(* IEC 61131-3 sources: SRCI/RobotLibrary/Library/POUs/_internal/BaseFBs, 4 files *)

(* ---- RobotLibraryBaseEnableFB.st ---- *)
FUNCTION_BLOCK RobotLibraryBaseEnableFB EXTENDS RobotLibraryBaseFB
// -------------------------------------------------------------------------
//  SRCI Robot Library
// -------------------------------------------------------------------------
//
//  Object:      RobotLibraryBaseFB
//  Author:      Thorsten Brach
//  Date:        2024-08-11
//
//  Description:
//
//
//  Copyright:
//    (C) 2024 Thorsten Brach. All rights reserved
//             Licensed under the LGPL-3.0 license.
//
//  Disclaimer:
//    This project is provided without any guarantee and can be used for
//    private and commercial purposes. Any use is at the user’s
//    own risk and responsibility.
//
// -------------------------------------------------------------------------
VAR_INPUT
  /// Set TRUE to activate / Set False to deactivate
  Enable            : BOOL;
END_VAR

VAR_OUTPUT
  /// FB is being processed
  Busy              : BOOL;
  /// TRUE while function is active
  Enabled           : BOOL;
END_VAR

VAR
  /// Rising edge for enable
  {attribute 'hide'}
 _enable_R          : R_TRIG;
  /// Falling edge for enable
  {attribute 'hide'}
 _enable_F          : F_TRIG;
END_VAR

  SUPER^(AxesGroup := AxesGroup);

END_FUNCTION_BLOCK

METHOD PROTECTED OnCall
VAR_IN_OUT
  /// Robot assignment of function
  AxesGroup : AxesGroup;
END_VAR

VAR
  /// internal return value
 _retVal : DINT;
END_VAR

  SUPER^.OnCall(AxesGroup := AxesGroup);

  // building rising and falling edges
  _enable_R( CLK := Enable);
  _enable_F( CLK := Enable);

  // Check command execution is allowed ?
  IF ((     Enable                                 ) AND
      ( NOT AxesGroup.State.Initialized            ) AND
      ( NOT AxesGroup.State.Synchronized           ) AND
      (     MyType <> 'MC_ExchangeConfigurationFB' ) AND // is part of init sequence
      (     MyType <> 'MC_ReadMessagesFB'          ) AND // is part of init sequence
      (     MyType <> 'MC_ReadRobotDataFB'         ))    // is part of init sequence
  THEN
    ErrorID := RobotLibraryErrorIdEnum.ERR_COMMANDS_NOT_ENABLED;
    Error   := TRUE;
    Busy    := FALSE;
  END_IF

  // On execution started
  IF ( _enable_R.Q )
  THEN
    OnExecStart(AxesGroup := AxesGroup);
  END_IF

  // On execution cancel
  IF ( Busy ) AND ( _enable_F.Q )
  THEN
    // set cancel flag
   _cancel := TRUE;
  END_IF

  IF ( _cancel )
  THEN
    // call Cancel
   _retVal := OnExecCancel(AxesGroup := AxesGroup);

    // done or error ?
    IF ( _retVal <> RobotLibraryConstants.RUNNING )
    THEN
      // reset cancel flag
     _cancel := FALSE;
  	END_IF
  END_IF

  // On execution error clear
  IF ( Error ) AND ( _enable_F.Q )
  THEN
    // set ClearError flag
   _clearError := TRUE;
  END_IF

  IF ( _clearError )
  THEN
   _retVal := OnExecErrorClear(AxesGroup := AxesGroup);

    // done or error ?
    IF ( _retVal <> RobotLibraryConstants.RUNNING )
    THEN
      // reset ClearError flag
     _clearError := FALSE;
  	END_IF
  END_IF

END_METHOD

METHOD Protected OnExecCancel : DINT
VAR_IN_OUT
  /// Robot assignment of function
  AxesGroup : AxesGroup;
END_VAR
VAR
  /// internal return value
 _retVal    : DINT;
END_VAR

  OnExecCancel := Reset();

  // Create log entry
  CreateLogMessagePara1 ( Timestamp   := AxesGroup.State.SystemTime,
                          MessageType := MessageType.CMD,
                          Severity    := Severity.DEBUG,
                          MessageCode := 0,
                          MessageText := 'Execution of {1} cancled ',
                          Para1       := MyType);

  // try to remove cmd
  _retVal := AxesGroup.Acyclic.ActiveCommandRegister.RemoveCmd(_uniqueID);

  IF (_retVal = RobotLibraryConstants.OK)
  THEN
    // Create log entry
    CreateLogMessagePara1 ( Timestamp   := AxesGroup.State.SystemTime,
                            MessageType := MessageType.CMD,
                            Severity    := Severity.DEBUG,
                            MessageCode := 0,
                            MessageText := '{1} successfully removed from ACR',
                            Para1       := MyType);
  ELSE
    // Create log entry
    CreateLogMessagePara1 ( Timestamp   := AxesGroup.State.SystemTime,
                            MessageType := MessageType.CMD,
                            Severity    := Severity.DEBUG,
                            MessageCode := 0,
                            MessageText := '{1} was not removed from ACR because execution was already in progress',
                            Para1       := MyType);
  END_IF

END_METHOD

METHOD PROTECTED OnExecErrorClear : DINT
VAR_IN_OUT
  /// Robot assignment of function
  AxesGroup : AxesGroup;
END_VAR

  OnExecErrorClear := RobotLibraryConstants.RUNNING;

  CASE _stepClearError OF

    0:  // Reset
        Reset();
        // trigger parameter update to disable FB
       _parameterUpdateInternal := TRUE;
        // call Check Parameter changed method to trigger the parameter update to deactivate jogging mode
        CheckParameterChanged(AxesGroup := AxesGroup);
        // set timeout
        SetTimeout(PT := _timeoutClearError, rTimer := _timerClearError);
        // inc step counter
       _stepClearError := _stepClearError + 1;

    1: IF ( _responseReceived )
       THEN
         // reset response received flag
        _responseReceived := FALSE;
         // reset step counter
        _stepClearError := 0;
         // finished
         OnExecErrorClear := RobotLibraryConstants.OK;
       ELSE
         // timeout exceeded ?
         IF (CheckTimeout(_timerClearError) = RobotLibraryConstants.OK)
         THEN
           OnExecErrorClear := RobotLibraryConstants.HAS_ERROR;
         END_IF
  	   END_IF
  ELSE
    // invalid step
    ErrorID := RobotLibraryErrorIdEnum.ERR_INVALID_STEP;
  END_CASE

  // reset step counter
  IF (OnExecErrorClear <> RobotLibraryConstants.RUNNING)
  THEN
   _stepClearError := 0;
  END_IF

END_METHOD

METHOD PROTECTED OnExecRun : DINT
VAR_IN_OUT
  /// Robot assignment of function
  AxesGroup : AxesGroup;
END_VAR

END_METHOD

METHOD PROTECTED OnExecStart : DINT
VAR_IN_OUT
  /// Robot assignment of function
  AxesGroup : AxesGroup;
END_VAR

END_METHOD

METHOD PROTECTED Reset : DINT
VAR_INPUT
END_VAR

  Reset := SUPER^.Reset();

  Busy    := FALSE;
  Enabled := FALSE;

END_METHOD

(* ---- RobotLibraryBaseExecuteFB.st ---- *)
FUNCTION_BLOCK RobotLibraryBaseExecuteFB EXTENDS RobotLibraryBaseFB
// -------------------------------------------------------------------------
//  SRCI Robot Library
// -------------------------------------------------------------------------
//
//  Object:      RobotLibraryBaseFB
//  Author:      Thorsten Brach
//  Date:        2024-08-11
//
//  Description:
//
//
//  Copyright:
//    (C) 2024 Thorsten Brach. All rights reserved
//             Licensed under the LGPL-3.0 license.
//
//  Disclaimer:
//    This project is provided without any guarantee and can be used for
//    private and commercial purposes. Any use is at the user’s
//    own risk and responsibility.
//
// -------------------------------------------------------------------------
VAR_INPUT
  /// Start of the command at the rising edge
  Execute         : BOOL;
END_VAR
VAR_OUTPUT
  /// The command has been completed successfully
  Done            : BOOL;
  /// FB is being processed
  Busy            : BOOL;
  /// Command is transferred and confirmed by the RC
//  CommandBuffered : BOOL;
END_VAR

VAR
  /// Rising edge for execute
  {attribute 'hide'}
 _execute_R       : R_TRIG;
  /// Falling edge for execute
  {attribute 'hide'}
 _execute_F       : F_TRIG;
END_VAR

  SUPER^(AxesGroup := AxesGroup);

END_FUNCTION_BLOCK

// Base implementation must be called !
METHOD PROTECTED OnCall
VAR_IN_OUT
  /// Robot assignment of function
  AxesGroup         : AxesGroup;
END_VAR

VAR
  /// internal return value
 _retVal : DINT;
END_VAR

  SUPER^.OnCall(AxesGroup := AxesGroup);

  // building rising and falling edges
  _execute_R( CLK := Execute);
  _execute_F( CLK := Execute);

  // Check command execution is allowed ?
  IF ((     Execute                                ) AND
      ( NOT AxesGroup.State.CMDsEnabled            ) AND
      (     MyType <> 'MC_ExchangeConfigurationFB' ) AND // is part of init sequence
      (     MyType <> 'MC_ReadMessagesFB'          ) AND // is part of init sequence
      (     MyType <> 'MC_ReadRobotDataFB'         ))    // is part of init sequence
  THEN
    ErrorID := RobotLibraryErrorIdEnum.ERR_COMMANDS_NOT_ENABLED;
    Error   := TRUE;
    Busy    := FALSE;
  END_IF

  // On execution started
  IF ( _execute_R.Q )
  THEN
    OnExecStart(AxesGroup := AxesGroup);
  END_IF

  // On execution cancel
  IF ( Busy ) AND ( _execute_F.Q )
  THEN
    // set cancel flag
   _cancel := TRUE;
  END_IF

  IF ( _cancel )
  THEN
    // call Cancel
   _retVal := OnExecCancel(AxesGroup := AxesGroup);

    // done or error ?
    IF ( _retVal <> RobotLibraryConstants.RUNNING )
    THEN
      // reset cancel flag
     _cancel := FALSE;
  	END_IF
  END_IF

  // On execution error clear
  IF ( Error ) AND ( _execute_F.Q )
  THEN
    // set ClearError flag
   _clearError := TRUE;
  END_IF

  IF ( _clearError )
  THEN
   _retVal := OnExecErrorClear(AxesGroup := AxesGroup);

    // done or error ?
    IF ( _retVal <> RobotLibraryConstants.RUNNING )
    THEN
      // reset ClearError flag
     _clearError := FALSE;
  	END_IF
  END_IF

END_METHOD

METHOD PROTECTED OnExecCancel : DINT
VAR_IN_OUT
  /// Robot assignment of function
  AxesGroup : AxesGroup;
END_VAR
VAR
  /// internal return value
 _retVal    : DINT;
END_VAR

  // Create log entry
  CreateLogMessagePara1 ( Timestamp   := AxesGroup.State.SystemTime,
                          MessageType := MessageType.CMD,
                          Severity    := Severity.DEBUG,
                          MessageCode := 0,
                          MessageText := 'Execution of {1} cancled ',
                          Para1       := MyType);

  // try to remove cmd
  _retVal := AxesGroup.Acyclic.ActiveCommandRegister.RemoveCmd(_uniqueID);

  IF (_retVal = RobotLibraryConstants.OK)
  THEN
    // Create log entry
    CreateLogMessagePara1 ( Timestamp   := AxesGroup.State.SystemTime,
                            MessageType := MessageType.CMD,
                            Severity    := Severity.DEBUG,
                            MessageCode := 0,
                            MessageText := '{1} successfully removed from ACR',
                            Para1       := MyType);
  ELSE
    // Create log entry
    CreateLogMessagePara1 ( Timestamp   := AxesGroup.State.SystemTime,
                            MessageType := MessageType.CMD,
                            Severity    := Severity.DEBUG,
                            MessageCode := 0,
                            MessageText := '{1} was not removed from ACR because execution was already in progress',
                            Para1       := MyType);
  END_IF

  OnExecCancel := Reset();

END_METHOD

METHOD PROTECTED OnExecErrorClear : DINT
VAR_IN_OUT
  /// Robot assignment of function
  AxesGroup : AxesGroup;
END_VAR

  OnExecErrorClear := Reset();

END_METHOD

METHOD PROTECTED OnExecRun : DINT
VAR_IN_OUT
  /// Robot assignment of function
  AxesGroup : AxesGroup;
END_VAR

END_METHOD

METHOD PROTECTED OnExecStart : DINT
VAR_IN_OUT
  /// Robot assignment of function
  AxesGroup : AxesGroup;
END_VAR

END_METHOD

METHOD PROTECTED Reset : DINT
VAR_INPUT
END_VAR

  Reset := SUPER^.Reset();

  Done := FALSE;
  Busy := FALSE;

END_METHOD

(* ---- RobotLibraryBaseFB.st ---- *)
FUNCTION_BLOCK RobotLibraryBaseFB EXTENDS RobotLibraryLogFB
// -------------------------------------------------------------------------
//  SRCI Robot Library
// -------------------------------------------------------------------------
//
//  Object:      RobotLibraryBaseFB
//  Author:      Thorsten Brach
//  Date:        2024-06-01
//
//  Description:
//
//
//  Copyright:
//    (C) 2024 Thorsten Brach. All rights reserved
//             Licensed under the LGPL-3.0 license.
//
//  Disclaimer:
//    This project is provided without any guarantee and can be used for
//    private and commercial purposes. Any use is at the user’s
//    own risk and responsibility.
//
// -------------------------------------------------------------------------
VAR_INPUT
  /// User defined command name
  Name         : STRING(80);
  /// Execution Mode
  ExecMode     : ExecutionMode;
  /// Priority
  Priority     : PriorityLevel;
END_VAR
VAR_OUTPUT
  /// Command data
  CommandData  : RobotLibraryCommandDataFB;
  /// response data
  ResponseData : RobotLibraryResponseDataFB;
  /// An error occurred during the execution of the command
  Error        : BOOL;
  /// ErrorID reported by RC for error identification according to Table 7-1
  ErrorID      : WORD;
  ErrorIdEnum  : RobotLibraryErrorIdEnum;
  ErrorAddTxt  : STRING(RobotLibraryConstants.MAX_ADD_TEXT_LENGTH);

  /// WarningID for warning identification reported during execution of command according to Table 7-3
  WarningID    : WORD;
  WarningIdEnum: RobotLibraryWarningIdEnum;
  /// InfoID for info identification reported during execution of command according to Table 7-5
  InfoID       : WORD;
  InfoIdEnum   : RobotLibraryInfoIdEnum;
END_VAR
VAR_IN_OUT
  /// Robot assignment of function
  AxesGroup    : AxesGroup;
END_VAR

VAR
  /// Rising edge for error
  {attribute 'hide'}
 _error_R                  : R_TRIG;
  /// Rising edge for warning
  {attribute 'hide'}
 _warning_R                : R_TRIG;
  /// Rising edge for information
  {attribute 'hide'}
 _info_R                   : R_TRIG;
  /// clear error active
 _clearError               : BOOL;
  /// cancel active
 _cancel                   : BOOL;
  /// unique ID
 _uniqueID                 : UDINT;
  /// flag for response received
 _responseReceived         : BOOL;
  /// internal step counter
 _stepCmd                  : DINT;
  /// internal timer
  {attribute 'hide'}
 _timerCmd                 : TON;
  /// internal timeout
  {attribute 'hide'}
 _timeoutCmd               : TIME := T#5S;
  /// internal step counter for ClearError
 _stepClearError           : DINT;
  /// internal timer for ClearError
  {attribute 'hide'}
 _timerClearError          : TON;
  /// internal timeout for ClearError
  {attribute 'hide'}
 _timeoutClearError        : TIME := T#5S;

  /// internal step counter for Cancel
 _stepCancel               : DINT;
  /// internal timer for Cancel
  {attribute 'hide'}
 _timerCancel              : TON;
  /// internal timeout for Cancel
  {attribute 'hide'}
 _timeoutCancel            : TIME := T#5S;

  /// internal command header
 _cmdHeader                : CmdHeader;
  /// internal response header
 _rspHeader                : RspHeader;
  /// internal flag for send a parameter update
 _parameterUpdateInternal  : BOOL;
  /// internal flag for parameter has changed
 _parameterChanged         : BOOL;
  /// internal flag for parameter are valid
 _parameterValid           : BOOL;
END_VAR

  OnCall               (AxesGroup := AxesGroup);
  OnExecRun            (AxesGroup := AxesGroup);
  CheckParameterChanged(AxesGroup := AxesGroup);

  IF ( AxesGroup.State.OnlineChange_R.Q )
  THEN
    OnOnlineChange(AxesGroup := AxesGroup);
  END_IF

END_FUNCTION_BLOCK

METHOD PUBLIC CallBack : DINT
VAR_INPUT
  /// Response data
  RspData   : AxesGroupAcyclicAcrEntryRspBuffer;
  /// Timestamp
  Timestamp : SystemTime;
END_VAR

  // Create log entry
  CreateLogMessagePara2 ( Timestamp   := Timestamp,
                          MessageType := MessageType.CMD,
                          Severity    := Severity.DEBUG,
                          MessageCode := 0,
                          MessageText := 'Callback reveiced in FB {1} <{2}>',
                          Para1       := MyType,
                          Para2       := Name);

  ResponseData.Reset();
  ResponseData.Payload    := RspData.Payload;
  ResponseData.PayloadLen := RspData.PayloadLen;
  ParseResponsePayload( ResponseData :=  ResponseData , Timestamp := Timestamp);

  // set flag for response received
  _responseReceived := TRUE;

END_METHOD

METHOD PROTECTED CheckFunctionSupported : BOOL
VAR_IN_OUT
  /// Robot assignment of function
  AxesGroup : AxesGroup;
END_VAR

  Error       := TRUE;
  ErrorID     := RobotLibraryErrorIdEnum.ERR_FUNCTION_NOT_SUPPORTED;
  ErrorAddTxt := CONCAT(THIS^._myType, ' ');
  ErrorAddTxt := CONCAT(ErrorAddTxt , THIS^.Name);

  // Create log entry
  CreateLogMessagePara1 ( Timestamp   := AxesGroup.State.SystemTime,
                          MessageType := MessageType.CMD,
                          Severity    := Severity.DEBUG,
                          MessageCode := 0,
                          MessageText := 'Execution canceled, because function <{1}> is not supported by the robot controller',
                          Para1       :=  _myType);

END_METHOD

METHOD PROTECTED CheckParameterChanged : BOOL
VAR_IN_OUT
  /// Robot assignment of function
  AxesGroup    : AxesGroup;
END_VAR

  IF ( CheckParameterChanged )
  THEN
    AxesGroup.Acyclic.ActiveCommandRegister.NotifyParameterChanged := _uniqueID;
  END_IF

END_METHOD

METHOD PROTECTED CheckParameterValid : BOOL
VAR_IN_OUT
  /// Robot assignment of function
  AxesGroup : AxesGroup;
END_VAR

  CheckParameterValid := TRUE;

END_METHOD

METHOD INTERNAL CreateCommandPayload : RobotLibraryCommandDataFB
VAR_IN_OUT
  /// Robot assignment of function
  AxesGroup    : AxesGroup;
END_VAR

  // Reset all variables
  CreateCommandPayload.Reset();
  // Add CmdType
  CreateCommandPayload.AddUint(_cmdHeader.CmdTyp);
  // Add Reserve_ExecMode
  CreateCommandPayload.AddHalfBytes(  0               , _cmdHeader.ExecMode);
  // Add ParSeq_Priority
  CreateCommandPayload.AddHalfBytes( _cmdHeader.ParSeq, _cmdHeader.Priority);

END_METHOD

METHOD PROTECTED OnCall
VAR_IN_OUT
  /// Robot assignment of function
  AxesGroup : AxesGroup;
END_VAR

  // map numeric value to enum, so that the corresponding message text is directly shown by the tooltip
  ErrorIdEnum   := ErrorId;
  WarningIdEnum := WarningId;
  InfoIdEnum    := InfoId;

  Error := ErrorID <> RobotLibraryConstants.OK;

  InternalLogger   := AxesGroup.MessageLog;
  ExternalLogger   := AxesGroup.MessageLog.ExternalLogger;
  LogLevel         := AxesGroup.MessageLog.LogLevel;

  // building rising edges for error, warning, info number detected
  _error_R  ( CLK := ErrorID   <> RobotLibraryConstants.OK );
  _warning_R( CLK := WarningID <> RobotLibraryConstants.OK );
  _info_R   ( CLK := InfoID    <> RobotLibraryConstants.OK );

  // Log Command events to message log
  IF  ( LogLevel < _rspHeader.AlarmMessageSeverity ) AND
     (( _error_R  .Q                               ) OR
      ( _warning_R.Q                               ) OR
      ( _info_R   .Q                               ))
  THEN
    // Add command message to message buffer
    AxesGroup.MessageLog
      .AddMessageLogByParameter(  Timestamp   :=   AxesGroup.State.SystemTime,
                                  MessageType :=   MessageType.CMD,
                                  MessageCode :=  _rspHeader.AlarmMessageCode,
                                  MessageText :=   CONCAT(MyType, CONCAT(' : ' , MESSAGE_CODE_TO_STRING(_rspHeader.AlarmMessageCode))),
                                  Severity    :=  _rspHeader.AlarmMessageSeverity );
  END_IF

  IF ( _error_R.Q)
  THEN
    // Create log entry
    CreateLogMessagePara2 ( Timestamp   := AxesGroup.State.SystemTime,
                            MessageType := MessageType.CMD,
                            Severity    := Severity.DEBUG,
                            MessageCode := 0,
                            MessageText := 'Error with ID: 16#{1} in FB {2} received ',
                            Para1       := WORD_TO_STRING_HEX(ErrorID),
                            Para2       := MyType);
  END_IF

  IF ( _warning_R.Q)
  THEN
    // Create log entry
    CreateLogMessagePara2 ( Timestamp   := AxesGroup.State.SystemTime,
                            MessageType := MessageType.CMD,
                            Severity    := Severity.DEBUG,
                            MessageCode := 0,
                            MessageText := 'Warning with ID: 16#{1} in FB {2} received ',
                            Para1       := WORD_TO_STRING_HEX(WarningID),
                            Para2       := MyType);
  END_IF

  IF ( _info_R.Q)
  THEN
    // Create log entry
    CreateLogMessagePara2 ( Timestamp   := AxesGroup.State.SystemTime,
                            MessageType := MessageType.CMD,
                            Severity    := Severity.DEBUG,
                            MessageCode := 0,
                            MessageText := 'Info with ID: 16#{1} in FB {2} received ',
                            Para1       := WORD_TO_STRING_HEX(InfoID),
                            Para2       := MyType);
  END_IF

END_METHOD

METHOD PROTECTED OnExecRun : DINT
VAR_IN_OUT
  /// Robot assignment of function
  AxesGroup : AxesGroup;
END_VAR

END_METHOD

METHOD OnOnlineChange : DINT
VAR_IN_OUT
  /// Robot assignment of function
  AxesGroup : AxesGroup;
END_VAR

  // update pointer to command FB
  AxesGroup.Acyclic.ActiveCommandRegister.OnOnlineChange( UniqueID := _uniqueID, pCommandFB := ADR(THIS^));

END_METHOD

METHOD INTERNAL ParseResponsePayload : DINT
VAR_INPUT
  /// Response data
  ResponseData : RobotLibraryResponseDataFB;
  /// Timestamp
  Timestamp    : SystemTime;
END_VAR

  // reset message IDs
  InfoID    := 0;
  WarningID := 0;
  ErrorID   := 0;

  // get State
  _rspHeader.State                := ResponseData.GetHalfeByte1(IncPayloadPtr := FALSE);
  // get ParSeq
  _rspHeader.ParSeq               := ResponseData.GetHalfeByte2(IncPayloadPtr := TRUE);
  // get AlarmMessageSeverity
  _rspHeader.AlarmMessageSeverity := ResponseData.GetSint();
  // get AlarmMessageCode
  _rspHeader.AlarmMessageCode     := ResponseData.GetUint();

  // Update InfoID / WarningID / ErrorID
  CASE _rspHeader.AlarmMessageSeverity OF

    // Informative message
    Severity.INFO        : InfoID    := _rspHeader.AlarmMessageCode;
    // Warning message
    Severity.WARNING     : WarningID := _rspHeader.AlarmMessageCode;
    // Error message
    Severity.ERROR       : ErrorID   := _rspHeader.AlarmMessageCode;
    // Fataö error message
    Severity.FATAL_ERROR : ErrorID   := _rspHeader.AlarmMessageCode;

  END_CASE

  ParseResponsePayload := ResponseData.PayloadPtr;

END_METHOD

METHOD PROTECTED Reset : DINT
VAR_INPUT
END_VAR

  _parameterUpdateInternal := FALSE;
  _responseReceived := FALSE;

  _uniqueId := 0;
  _stepCmd  := 0;
  Error     := FALSE;
  ErrorID   := 0;
  WarningID := 0;
  InfoID    := 0;

  Reset := RobotLibraryConstants.OK;

END_METHOD

(* ---- RobotLibraryLogFB.st ---- *)
FUNCTION_BLOCK RobotLibraryLogFB
// -------------------------------------------------------------------------
//  SRCI Robot Library
// -------------------------------------------------------------------------
//
//  Object:      RobotLibraryLogFB
//  Author:      Thorsten Brach
//  Date:        2024-11-10
//
//  Description:
//
//
//  Copyright:
//    (C) 2024 Thorsten Brach. All rights reserved
//             Licensed under the LGPL-3.0 license.
//
//  Disclaimer:
//    This project is provided without any guarantee and can be used for
//    private and commercial purposes. Any use is at the user’s
//    own risk and responsibility.
//
// -------------------------------------------------------------------------
VAR_INPUT
  /// Interface to an internal logger
  InternalLogger : IMessageLogger;
  /// Interface to an external logger
  ExternalLogger : IMessageLogger;
  /// Logging level
  LogLevel       : LogLevelEnum := LogLevelEnum.INFO;
END_VAR

VAR
  /// Type of the function block
 _myType         : STRING;
END_VAR

END_FUNCTION_BLOCK

METHOD CreateLogMessage : STRING(RobotLibraryParameter.MESSAGE_TEXT_LEN)
VAR_INPUT
  /// Timestamp
  Timestamp   : SystemTime;
  /// Type of message according to Table 5-46:
  MessageType : MessageType;
  /// Severity of message according to Table 5-47: Debug, Info, Warning, Error, Fatal error
  Severity    : Severity;
  /// Code of messages
  MessageCode : DWORD;
  /// Static text of message
  MessageText : STRING(RobotLibraryParameter.MESSAGE_TEXT_LEN);
END_VAR

VAR
  /// internal log message
 _message    : AlarmMessage;
  /// internal string
 _tmpString  : STRING(255);
END_VAR

  IF ( LogLevel <= Severity )
  THEN
   _message.Timestamp   := Timestamp;
   _message.MessageType := MessageType;
   _message.Severity    := Severity;
   _message.MessageCode := MessageCode;
   _message.MessageText := StrPadRight(MyType,' ', RobotLibraryDefines.MaxTypeNameLength);
   _message.MessageText := CONCAT(_message.MessageText, ': ');
   _message.MessageText := CONCAT(_message.MessageText,MessageText);

    // return log message
    CreateLogMessage := ALARM_MESSAGE_TO_STRING(_message);

    // Check internal logger valid ?
    IF ( InternalLogger <> 0 )
    THEN
      InternalLogger.AddSystemLog( SystemLog := ALARM_MESSAGE_TO_STRING(_message));
    END_IF

    // Check external logger valid ?
    IF ( ExternalLogger <> 0 )
    THEN
      ExternalLogger.AddSystemLog( SystemLog := ALARM_MESSAGE_TO_STRING(_message));
    END_IF
  END_IF

END_METHOD

METHOD CreateLogMessagePara1 : STRING(RobotLibraryParameter.MESSAGE_TEXT_LEN)
VAR_INPUT
  /// Timestamp
  Timestamp   : SystemTime;
  /// Type of message according to Table 5-46:
  MessageType : MessageType;
  /// Severity of message according to Table 5-47: Debug, Info, Warning, Error, Fatal error
  Severity    : Severity;
  /// Code of messages
  MessageCode : DWORD;
  /// Static text of message
  MessageText : STRING(RobotLibraryParameter.MESSAGE_TEXT_LEN);
  /// sub string which will replace the placeholder {1}
  Para1       : STRING(RobotLibraryParameter.MESSAGE_TEXT_LEN);
END_VAR
VAR
  /// internal log message
 _logMessage : AlarmMessage;
END_VAR

  IF ( LogLevel <= Severity )
  THEN
    MessageText := StrReplace(MessageText,'{1}', Para1);

    CreateLogMessagePara1
      := CreateLogMessage( Timestamp   := Timestamp,
                           MessageType := MessageType,
                           Severity    := Severity,
                           MessageCode := MessageCode,
                           MessageText := MessageText);
  END_IF

END_METHOD

METHOD CreateLogMessagePara2 : STRING(RobotLibraryParameter.MESSAGE_TEXT_LEN)
VAR_INPUT
  /// Timestamp
  Timestamp   : SystemTime;
  /// Type of message according to Table 5-46:
  MessageType : MessageType;
  /// Severity of message according to Table 5-47: Debug, Info, Warning, Error, Fatal error
  Severity    : Severity;
  /// Code of messages
  MessageCode : DWORD;
  /// Static text of message
  MessageText : STRING(RobotLibraryParameter.MESSAGE_TEXT_LEN);
  /// sub string which will replace the placeholder {1}
  Para1       : STRING(RobotLibraryParameter.MESSAGE_TEXT_LEN);
  /// sub string which will replace the placeholder {2}
  Para2       : STRING(RobotLibraryParameter.MESSAGE_TEXT_LEN);
END_VAR
VAR
  /// internal log message
 _logMessage : AlarmMessage;
END_VAR

  IF ( LogLevel <= Severity )
  THEN
    MessageText := StrReplace(MessageText,'{2}', Para2);

    CreateLogMessagePara2
      := CreateLogMessagePara1( Timestamp   := Timestamp,
                                MessageType := MessageType,
                                Severity    := Severity,
                                MessageCode := MessageCode,
                                MessageText := MessageText,
                                Para1       := Para1);
  END_IF

END_METHOD

METHOD CreateLogMessagePara3 : STRING(RobotLibraryParameter.MESSAGE_TEXT_LEN)
VAR_INPUT
  /// Timestamp
  Timestamp   : SystemTime;
  /// Type of message according to Table 5-46:
  MessageType : MessageType;
  /// Severity of message according to Table 5-47: Debug, Info, Warning, Error, Fatal error
  Severity    : Severity;
  /// Code of messages
  MessageCode : DWORD;
  /// Static text of message
  MessageText : STRING(RobotLibraryParameter.MESSAGE_TEXT_LEN);
  /// sub string which will replace the placeholder {1}
  Para1       : STRING(RobotLibraryParameter.MESSAGE_TEXT_LEN);
  /// sub string which will replace the placeholder {2}
  Para2       : STRING(RobotLibraryParameter.MESSAGE_TEXT_LEN);
  /// sub string which will replace the placeholder {3}
  Para3       : STRING(RobotLibraryParameter.MESSAGE_TEXT_LEN);
END_VAR
VAR
  /// internal log message
 _logMessage : AlarmMessage;
END_VAR

  IF ( LogLevel <= Severity )
  THEN
    MessageText := StrReplace(MessageText,'{3}', Para3);

    CreateLogMessagePara3
      := CreateLogMessagePara2( Timestamp   := Timestamp,
                                MessageType := MessageType,
                                Severity    := Severity,
                                MessageCode := MessageCode,
                                MessageText := MessageText,
                                Para1       := Para1,
                                Para2       := Para2);
  END_IF

END_METHOD

METHOD CreateLogMessagePara4 : STRING(RobotLibraryParameter.MESSAGE_TEXT_LEN)
VAR_INPUT
  /// Timestamp
  Timestamp   : SystemTime;
  /// Type of message according to Table 5-46:
  MessageType : MessageType;
  /// Severity of message according to Table 5-47: Debug, Info, Warning, Error, Fatal error
  Severity    : Severity;
  /// Code of messages
  MessageCode : DWORD;
  /// Static text of message
  MessageText : STRING(RobotLibraryParameter.MESSAGE_TEXT_LEN);
  /// sub string which will replace the placeholder {1}
  Para1       : STRING(RobotLibraryParameter.MESSAGE_TEXT_LEN);
  /// sub string which will replace the placeholder {2}
  Para2       : STRING(RobotLibraryParameter.MESSAGE_TEXT_LEN);
  /// sub string which will replace the placeholder {3}
  Para3       : STRING(RobotLibraryParameter.MESSAGE_TEXT_LEN);
  /// sub string which will replace the placeholder {4}
  Para4       : STRING(RobotLibraryParameter.MESSAGE_TEXT_LEN);
END_VAR
VAR
  /// internal log message
 _logMessage : AlarmMessage;
END_VAR

  IF ( LogLevel <= Severity )
  THEN
    MessageText := StrReplace(MessageText,'{4}', Para4);

    CreateLogMessagePara4
      := CreateLogMessagePara3( Timestamp   := Timestamp,
                                MessageType := MessageType,
                                Severity    := Severity,
                                MessageCode := MessageCode,
                                MessageText := MessageText,
                                Para1       := Para1,
                                Para2       := Para2,
                                Para3       := Para3);
  END_IF

END_METHOD

METHOD CreateLogMessagePara5 : STRING(RobotLibraryParameter.MESSAGE_TEXT_LEN)
VAR_INPUT
  /// Timestamp
  Timestamp   : SystemTime;
  /// Type of message according to Table 5-46:
  MessageType : MessageType;
  /// Severity of message according to Table 5-47: Debug, Info, Warning, Error, Fatal error
  Severity    : Severity;
  /// Code of messages
  MessageCode : DWORD;
  /// Static text of message
  MessageText : STRING(RobotLibraryParameter.MESSAGE_TEXT_LEN);
  /// sub string which will replace the placeholder {1}
  Para1       : STRING(RobotLibraryParameter.MESSAGE_TEXT_LEN);
  /// sub string which will replace the placeholder {2}
  Para2       : STRING(RobotLibraryParameter.MESSAGE_TEXT_LEN);
  /// sub string which will replace the placeholder {3}
  Para3       : STRING(RobotLibraryParameter.MESSAGE_TEXT_LEN);
  /// sub string which will replace the placeholder {4}
  Para4       : STRING(RobotLibraryParameter.MESSAGE_TEXT_LEN);
  /// sub string which will replace the placeholder {5}
  Para5       : STRING(RobotLibraryParameter.MESSAGE_TEXT_LEN);
END_VAR
VAR
  /// internal log message
 _logMessage : AlarmMessage;
END_VAR

  IF ( LogLevel <= Severity )
  THEN
    MessageText := StrReplace(MessageText,'{5}', Para5);

    CreateLogMessagePara5
      := CreateLogMessagePara4( Timestamp   := Timestamp,
                                MessageType := MessageType,
                                Severity    := Severity,
                                MessageCode := MessageCode,
                                MessageText := MessageText,
                                Para1       := Para1,
                                Para2       := Para2,
                                Para3       := Para3,
                                Para4       := Para4);
  END_IF

END_METHOD

METHOD CreateLogMessagePara6 : STRING(RobotLibraryParameter.MESSAGE_TEXT_LEN)
VAR_INPUT
  /// Timestamp
  Timestamp   : SystemTime;
  /// Type of message according to Table 5-46:
  MessageType : MessageType;
  /// Severity of message according to Table 5-47: Debug, Info, Warning, Error, Fatal error
  Severity    : Severity;
  /// Code of messages
  MessageCode : DWORD;
  /// Static text of message
  MessageText : STRING(RobotLibraryParameter.MESSAGE_TEXT_LEN);
  /// sub string which will replace the placeholder {1}
  Para1       : STRING(RobotLibraryParameter.MESSAGE_TEXT_LEN);
  /// sub string which will replace the placeholder {2}
  Para2       : STRING(RobotLibraryParameter.MESSAGE_TEXT_LEN);
  /// sub string which will replace the placeholder {3}
  Para3       : STRING(RobotLibraryParameter.MESSAGE_TEXT_LEN);
  /// sub string which will replace the placeholder {4}
  Para4       : STRING(RobotLibraryParameter.MESSAGE_TEXT_LEN);
  /// sub string which will replace the placeholder {5}
  Para5       : STRING(RobotLibraryParameter.MESSAGE_TEXT_LEN);
  /// sub string which will replace the placeholder {6}
  Para6       : STRING(RobotLibraryParameter.MESSAGE_TEXT_LEN);
END_VAR
VAR
  /// internal log message
 _logMessage : AlarmMessage;
END_VAR

  IF ( LogLevel <= Severity )
  THEN
    MessageText := StrReplace(MessageText,'{6}', Para6);

    CreateLogMessagePara6
      := CreateLogMessagePara5( Timestamp   := Timestamp,
                                MessageType := MessageType,
                                Severity    := Severity,
                                MessageCode := MessageCode,
                                MessageText := MessageText,
                                Para1       := Para1,
                                Para2       := Para2,
                                Para3       := Para3,
                                Para4       := Para4,
                                Para5       := Para5);
  END_IF

END_METHOD

PROPERTY PROTECTED MyType : STRING

GET
VAR
END_VAR

  MyType := _myType;

END_GET

SET
VAR
END_VAR

  _myType := MyType;

  // set the max type name length
  RobotLibraryDefines.MaxTypeNameLength := MAX(LEN(_myType), RobotLibraryDefines.MaxTypeNameLength);

END_SET
